// TwinCAT 3 PLC project StudentStation
// ProgramVersion: 3.1.4022.4
// libraries:
//   Tc2_Standard, * (Beckhoff Automation GmbH)
//   Tc2_System, * (Beckhoff Automation GmbH)
//   Tc3_Module, * (Beckhoff Automation GmbH)
//   VisuDialogs, * (System)
//   VisuSymbols,3.5.10.0,System
// project tree:
//   ABBControl/ ABBAssemble.TcPOU (not stored), ABBGotoAGVPos.TcPOU (not stored), ABBGotoBuffer.TcPOU (not stored), ABBGotoHome.TcPOU (not stored), ABBGotoScanner.TcPOU (not stored), ABBGotoTable.TcPOU (not stored), ABBPickLeaveBuffer.TcPOU (not stored), ABBPickLeaveContainerAGV.TcPOU (not stored), ABBPickLeaveContaineronTable.TcPOU (not stored), ABBPickLeaveScanner.TcPOU (not stored), ABBScanContainer.TcPOU (not stored), ABBScannerStation.TcPOU (not stored)
//   Automation Library/ AGVControlSystem.TcPOU (not stored), AutomationLibrary.TcPOU (not stored), BookingSystem.TcPOU (not stored), CommData.TcGVL (not stored), OrderHandling.TcPOU (not stored), PhysicalSystemTest.TcPOU (not stored), RobotControlSystem.TcPOU (not stored), RobotPosTracker.TcPOU (not stored), SensorReader.TcPOU (not stored), Visualaisation_Control.TcPOU (not stored)
//   DUTs/ ABBPositions.TcDUT (not stored), ABBXYPOS.TcDUT (not stored), OrderPLC.TcDUT (not stored), PLCRobotOrder.TcDUT (not stored), Station.TcDUT (not stored), Storage.TcDUT (not stored)
//   / GlobalTextList.TcGTLO (not stored), PlcTask.TcTTO (not stored), Visualization Manager.TcVMO (not stored)
//   GVLs/ GVL.TcGVL
//   POUs/ MAIN.TcPOU
//   VISUs/ RobotStation.TcVIS (not stored), Station.TcVIS, Visualization.TcVIS

// ---- GVLs/GVL.TcGVL
{attribute 'qualified_only'}
VAR_GLOBAL
	// Order for the next assembly part. The part name should be sent as per the part list and case sensitive. 
	{attribute 'OPC.UA.DA' := '1'}
	qsOrderFornextAssembly AT %Q*: STRING := '0';
	// Parts in your Station buffer. Each buffer have 3 storage locations. The part name and quantity should be mentioned.
	{attribute 'OPC.UA.DA' := '1'}
	BufferProducts AT %Q*: Station;
	// Signal to AGV, a pallet is placed from Station to the AGV. 
	{attribute 'OPC.UA.DA' := '1'}
	qxPalletPlacedinAGV AT %Q*: BOOL;
	// Signal From AGV, that it have docked in your station
	{attribute 'OPC.UA.DA' := '1'}
	ixAGVatStation AT %I*: BOOL;
	// Signal Denoting An AGV have arrived in the Station
	{attribute 'OPC.UA.DA' := '1'}	
	qxPickedfromAGV AT %Q*:BOOL; //Part is picked up from the AGV
	{attribute 'OPC.UA.DA' := '1'}
	mwStationStatus AT %Q*: INT; //Pre-Conditioning Mode //100:Ready to Work § 200: Getting Booked § 300: Booked and Busy § 400 : Manual mode  § 500: Pause Mode § 1000 : Emergency Mode 
	{attribute 'OPC.UA.DA' := '1'}	
	// Emergency Stop is active
	ixEmergencyStop AT %Q*:BOOL;
	
	// Inductive sensor reading. from scaning station
	ixInductiveSensor1 AT %I*:BOOL;
	// Inductive sensor reading. from scaning station
	ixInductiveSensor2 AT %I*:BOOL;
	// Inductive sensor reading. from scaning station
	ixInductiveSensor3 AT %I*:BOOL;
	// Inductive sensor reading. from scaning station
	ixInductiveSensor4 AT %I*:BOOL;
	// Inductive sensor reading. from the sensor in robot Tool
	ixInductiveSensorinTool AT %I*:BOOL;
	// Station ID of the station you are working with.
	{attribute 'OPC.UA.DA' := '1'}
	mwStationID AT %Q*: INT;
	
END_VAR

// ---- POUs/MAIN.TcPOU
PROGRAM MAIN
VAR
END_VAR

AutomationLibrary();
Visualaisation_Control();
RobotPosTracker();

END_PROGRAM

// ---- VISUs/Station.TcVIS
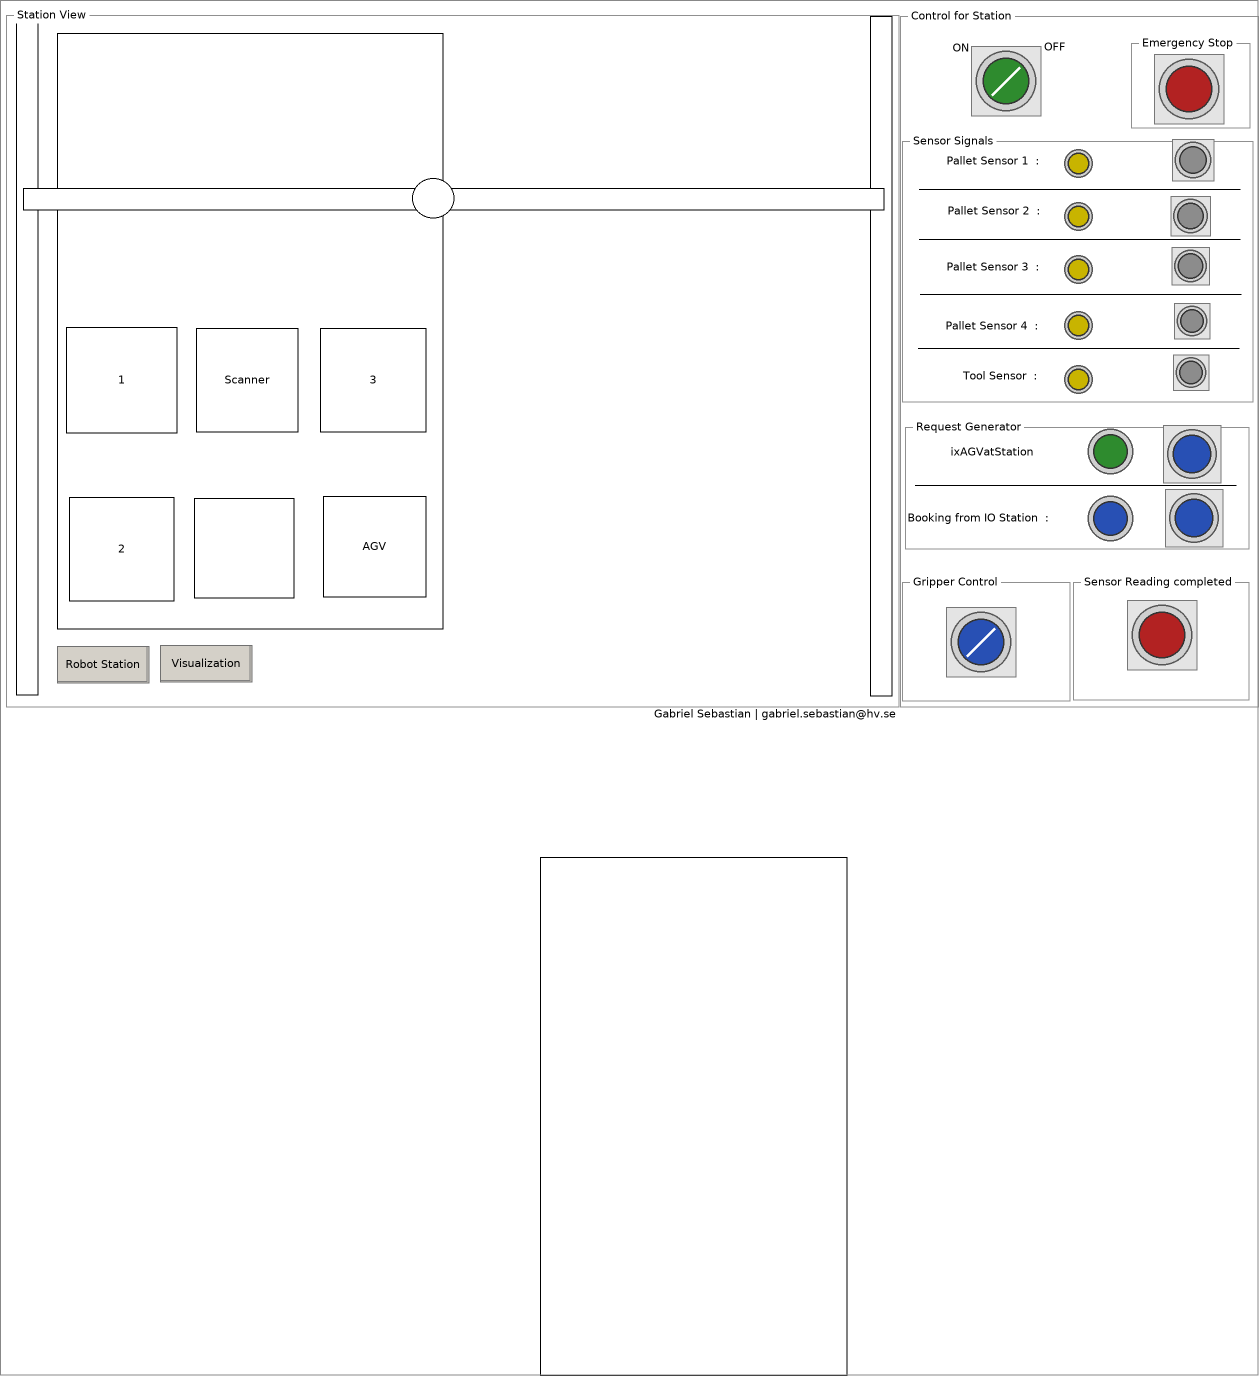
VISUALIZATION Station  // 1259x1376
    RoundedRectangle (540,857 307x519)
        p2738717112: CommData.mwCurrentAGVPOS
    Rectangle (16,15 22x680)
    GroupBox (6,7 893x700), "Station View"
        Rectangle (51,26 386x596)
        Rectangle (864,9 22x680)
        Rectangle (188,491 100x100)
        Rectangle (317,489 103x101), "AGV"
        Rectangle (190,321 102x104), "Scanner"
        Rectangle (60,320 111x106), "1"
        Rectangle (314,321 106x104), "3"
        Rectangle (63,490 105x104), "2"
        RoundedRectangle (17,181 861x22)
            p2738717112: CommData.mwYaxis
        Ellipse (406,171 42x40)
            p2738717112: CommData.mwYaxis
            p3560616238: CommData.mwXaxis
        Button (154,638 92x37), "Visualization"
            OnMouseClick: change screen: Visualization
        Button (51,639 92x37), "Robot Station"
            OnMouseClick: change screen: RobotStation
    GroupBox (900,8 359x699), "Control for Station"
        GroupBox (2,125 351x269), "Sensor Signals"
            Label (15,178 150x30), "Pallet Sensor 4 :"
            Label (17,63 150x30), "Pallet Sensor 2 :"
            Label (16,13 150x30), "Pallet Sensor 1 :"
            Line (17,56) (338,56)
            Lamp1 (160,14 33x33), variable: GVL.ixInductiveSensor1, style: Lamp-Lamp1-Yellow
            Lamp1 (160,67 33x33), variable: GVL.ixInductiveSensor2, style: Lamp-Lamp1-Yellow
            Lamp1 (160,120 33x33), variable: GVL.ixInductiveSensor3, style: Lamp-Lamp1-Yellow
            Lamp1 (160,176 33x33), variable: GVL.ixInductiveSensor4, style: Lamp-Lamp1-Yellow
            Label (16,119 150x30), "Pallet Sensor 3 :"
            Label (23,228 150x30), "Tool Sensor :"
            Lamp1 (160,230 33x33), variable: GVL.ixInductiveSensorinTool, style: Lamp-Lamp1-Yellow
            PushSwitch (266,6 50x42), variable: GVL.ixInductiveSensor1, input disabled if: CommData.mxRobotOnline, behaviour: TOGGLE, style: Switch-PushSwitch-Gray
            PushSwitch (267,63 43x40), variable: GVL.ixInductiveSensor2, input disabled if: CommData.mxRobotOnline, behaviour: TOGGLE, style: Switch-PushSwitch-Gray
            PushSwitch (269,114 39x38), variable: GVL.ixInductiveSensor3, input disabled if: CommData.mxRobotOnline, behaviour: TOGGLE, style: Switch-PushSwitch-Gray
            PushSwitch (270,170 40x36), variable: GVL.ixInductiveSensor4, input disabled if: CommData.mxRobotOnline, behaviour: TOGGLE, style: Switch-PushSwitch-Gray
            PushSwitch (271,221 36x37), variable: GVL.ixInductiveSensorinTool, input disabled if: CommData.mxRobotOnline, behaviour: TOGGLE, style: Switch-PushSwitch-Gray
            Line (17,106) (338,106)
            Line (18,161) (339,161)
            Line (16,215) (337,215)
        RotarySwitch (71,38 70x70), variable: CommData.mxOnlineMode, invisible if: CommData.mxRobotOnline, behaviour: TOGGLE, style: Switch-RotarySwitch-Green
        Label (106,24 98x30), "OFF", invisible if: CommData.mxRobotOnline
        Label (12,25 98x30), "ON", invisible if: CommData.mxRobotOnline
        GroupBox (5,411 344x130), "Request Generator"
            Label (12,18 150x30), "ixAGVatStation"
            Line (10,66) (331,66)
            Lamp1 (177,6 57x53), variable: CommData.mxRequestAGV, style: Lamp-Lamp1-Green
            PushSwitch (257,6 60x58), variable: GVL.ixAGVatStation, behaviour: TOGGLE, style: Switch-PushSwitch-Blue
            Lamp1 (177,73 57x53), variable: CommData.mxNewBookingrequest, style: Lamp-Lamp1-Blue
            PushSwitch (259,70 60x58), variable: CommData.mxNewBookingrequest, behaviour: TOGGLE, style: Switch-PushSwitch-Blue
        GroupBox (173,566 176x126), "Sensor Reading completed", invisible if: NOT CommData.mxWaitingforSensorinput
            PushSwitch (54,26 70x70), variable: CommData.mxScannernoobject, behaviour: TAP, style: Switch-PushSwitch-Red
        GroupBox (2,566 168x127), "Gripper Control"
            Lamp1 (-1748,-553 70x70), style: Lamp-Lamp1-Yellow
            Lamp1 (44,34 70x70), variable: CommData.mxGripper, style: Lamp-Lamp1-Yellow
            RotarySwitch (44,33 70x70), variable: CommData.mxGripper, invisible if: NOT Visualaisation_Control.mxManualMode, behaviour: TOGGLE, style: Switch-RotarySwitch-Blue
        GroupBox (231,27 119x93), "Emergency Stop"
            PushSwitch (23,19 70x70), variable: GVL.ixEmergencyStop, behaviour: TOGGLE, style: Switch-PushSwitch-Red
    Label (900,503 156x30), "Booking from IO Station :"
    Label (650,699 250x30), "Gabriel Sebastian | gabriel.sebastian@hv.se"
END_VISUALIZATION

// ---- VISUs/Visualization.TcVIS
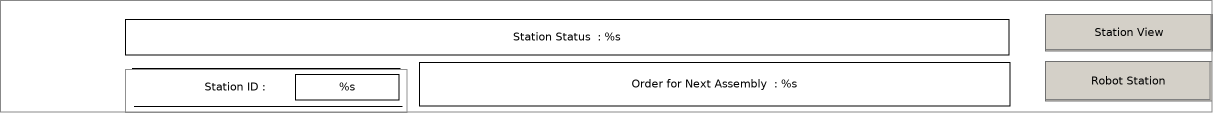
VISUALIZATION Visualization  // 1213x113
    Rectangle (125,19 884x36), "Station Status : %s", text variable: Visualaisation_Control.mxStationStatus
    GroupBox (125,61 282x52)
        Line (6,458) (274,458)
        Line (7,7) (275,7)
        Label (35,11 150x30), "Station ID :"
        Rectangle (170,13 104x26), "%s", text variable: GVL.mwStationID
        Line (9,45) (277,45)
    Button (1045,61 167x40), "Robot Station"
        OnMouseClick: change screen: RobotStation
    Rectangle (419,62 591x44), "Order for Next Assembly : %s", text variable: GVL.qsOrderFornextAssembly
    Button (1045,14 168x37), "Station View"
        OnMouseClick: change screen: Station
END_VISUALIZATION
